FUNCTION_BLOCK Outlet IMPLEMENTS I_Domain, I_Execute
VAR_INPUT
	bRequestButton	: BOOL;
END_VAR
VAR_OUTPUT
	bDrainValveOpen	: BOOL;
END_VAR
VAR CONSTANT
	MAX_STATE		: UDINT := 2;
END_VAR
VAR
	exe				: Execute(THIS^);

	// Context
	ctx				: Outlet_Ctx;

	// State Machine
	stateMachine	: StateMachine;
	stateRepo		: StateRepo<MAX_STATE>;
	stateBuffer		: StateBuffer<MAX_STATE>;
	stateMgr		: StateManager<MAX_STATE>(stateMachine, stateRepo, stateBuffer);
	A_Smgr			: A_StateManager(stateMgr, ctx.smgr);
	
	// States
	
	EStop			: Outlet_EStop(stateRepo, ctx);
	A_EStop			: A_Tag(EStop.Tag, ctx.iEStop);
	OnEStop			: Receiver(EStop);
	
	Operational		: Outlet_Operational(stateRepo, ctx);
	A_Operational	: A_Tag(Operational.Tag, ctx.iOperational);
	
	// FLAGS
	flagList		: FlagList<0>;
	
	// SIGNALS
	signalList		: SignalList<1>;
	A_SmgrChange	: A_Signal(signalList, stateMgr.GetOnChange());
	
	// RECEIVERS
	receiverList	: ReceiverList<1>;
	A_OnEStop		: A_Receiver(receiverList, OnEStop);
	
	// DOMAIN
	domTag			: Tag;
	domain			: Domain(domTag, stateMgr, flagList, signalList, receiverList);
	
	// PRIV
	bInit			: BOOL := TRUE;
END_VAR

METHOD AssignTank : Result
VAR_INPUT
	iTank		: I_Domain;
END_VAR
IF ctx.iIsEmpty <> 0 THEN
	AssignTank := None; // None is default, so this is not necessary!
	RETURN;
END_IF

IF iTank = 0 THEN
	AssignTank := Error;
	RETURN;
END_IF

ctx.iTank := iTank;

// Alternatively, this will carry over the error from inside the FindFlag function, 
// whereas the CASE option allows for change of error type.
(*
IF IsErr(FindFlag(iTank.Flags, 'IsEmpty', iFlag => ctx.iIsEmpty), eCarry => AssignTank) THEN
		DebugMsg(THIS^, 'Missing iIsEmpty! >');
		DebugMsg(iTank, '< Missing iIsEmpty!');
END_IF
*)

CASE FindFlag(iTank.Flags, 'IsEmpty', iFlag => ctx.iIsEmpty) OF 
	Error:
		DebugMsg(THIS^, 'Missing iIsEmpty! >');
		DebugMsg(iTank, '< Missing iIsEmpty!');
		
		AssignTank := Error;
	Ok:	
		AssignTank := Ok;
END_CASE
END_METHOD

METHOD Execute
IF bInit THEN
	ctx.smgr.Request(ctx.iOperational);

	bInit := FALSE;
END_IF

// INPUTS
ctx.bRequestButton := bRequestButton;

// OUTPUTS
bDrainValveOpen := ctx.bDrainValveOpen;
END_METHOD

PROPERTY Flags : Domains.Flags.I_FlagList
GET
Flags := flagList;
END_GET
END_PROPERTY

PROPERTY Recs : Domains.Broadcast.I_ReceiverList
GET
Recs := receiverList;
END_GET
END_PROPERTY

PROPERTY Signals : Domains.Broadcast.I_SignalList
GET
Signals := signalList;
END_GET
END_PROPERTY

PROPERTY Smgr : Domains.States.I_StateManager
GET
Smgr := stateMgr;
END_GET
END_PROPERTY

PROPERTY Tag : Tags.I_Tag
GET
Tag := domTag;
END_GET
END_PROPERTY

METHOD ToDebug : Debug.I_Debug
ToDebug := THIS^;
END_METHOD

END_FUNCTION_BLOCK

(* stored: Version 1.1.0.1
   POU Outlet: Id {08f78f88-2f7d-4896-98eb-be94062c7e0b}, SpecialFunc None
   Method AssignTank: Id {2b86b81f-cf6c-43cd-938d-bf9a462ab9fd}
   Method Execute: Id {ca2250aa-289a-487f-89bb-e08060846c74}
   Property Flags: Id {e882d9af-6ec0-434e-8b04-d89f6b7134df}
   Get Get: Id {ca52d541-87d6-4a9e-937f-7f63b72bdf08}
   Property Recs: Id {9063afe4-f19e-4025-878f-d63a2f9943b3}
   Get Get: Id {565d9f10-71df-4a7b-931d-ff80c27036cc}
   Property Signals: Id {ab4a53ab-2dc3-439b-ac7c-e9310c9aebba}
   Get Get: Id {66f8cabd-c820-4c3b-8a83-61a89d97672b}
   Property Smgr: Id {7eaf3a87-de67-47d9-b080-58ca0f216505}
   Get Get: Id {efe03c50-7ae2-4b7b-af46-43737d22c57e}
   Property Tag: Id {5202264c-6afa-4eb7-80cf-eda1e87ca599}
   Get Get: Id {c2474f0c-bd37-4dbc-a2eb-4d4bdc8c7aa3}
   Method ToDebug: Id {f9567eda-f289-4d30-af80-d3a880449631} *)
